(* CoDeSys 2.3.9.59 project: C2_Write_On_USB_or_SD.pro *)
(* Libraries: Standard.lib, Util.lib 20.3.15 10:30:08, SysLibCallback.lib, SysLibSockets.lib, SysLibTasks.lib, SysLibRtc.lib, SysLibFile.lib, SysLibPlcCtrl.lib *)

(* Task configuration *)
TASK tskMain (PRIORITY := 1, INTERVAL := T#20ms);
	MAIN();
END_TASK
TASK tskFiles (PRIORITY := 10, INTERVAL := T#100ms);
	prgCsvLogger();
END_TASK

(* Data type *)
TYPE stParameters :
STRUCT
	Start_stop	: BOOL;
	Temp1		: WORD;
	Temp2		: WORD;
	Temp3		: WORD;
END_STRUCT
END_TYPE

(* POU 10_Program/MAIN, ST *)
PROGRAM MAIN
VAR
	iCpt: INT := 0;
END_VAR
iCpt := iCpt + 1;
END_PROGRAM

(* POU 10_Program/prgCsvLogger, ST *)
PROGRAM prgCsvLogger
VAR
    Horodatage      : DT;					(* Horodate courante *)

    Trig            : R_TRIG;				(* Déclencheur montée *)
    Ligne           : fbStringBuilder;
    Texte           : STRING(255);
    NbOctets        : DWORD;

    xStart			: BOOL;					(* Impulsion externe de création fichier *)
    xDoItDone       : BOOL;					(* Flag interne d'état *)

    FileName        : STRING := '\InternalStorage\log_file.csv'; (* \InternalStorage ou \UsbStorage ou \StorageCard *)
    Fichier         : fbFileWriter;
    Bytes_Written   : DWORD;
    File_Size       : DWORD;
END_VAR
(*=================================================================================================
PROJET          : Data_To_CSV
DESCRIPTION     : Exemple générique de création et d'enregristement de données dans un 
                  fichier .csv stocké dans la mémoire interne du XV100 "/InternalStorage"
---------------------------------------------------------------------------------------------------
MATERIEL CIBLE  : XV102 (Adaptable à d'autres XV/XC en modifiant le path
LOGICIEL        : CODESYS V2.3.9 SP8
LIBRAIRIES      :
	- Standard.lib (V4.10.05) : R_TRIG
	- SysLibFile.lib (V23.9.04) : SysFileOpen, SysFileWrite, SysFileGetSize, SysFileClose

AUTEUR          : COTTANCIN Bruno
DATE            : 24/03/2026
VERSION         : V1.1.0

HISTORIQUE DES MODIFICATIONS :
---------------------------------------------------------------------------------------------------
V1.0.0 | 21/03/2026 | B. COTTANCIN | Création initiale (séquences, function blocks, etc.)
V1.0.1 | 22/03/2026 | B. COTTANCIN | Finalisation de l'architecture générale avant tests
V1.1.0 | 24/03/2026 | B. COTTANCIN | Commentaires FR + en-tête mis à jour

===================================================================================================
IMPORTANT                                 
===================================================================================================
CE PROGRAMME D'ECRITURE CSV DOIT IMPERATIVEMENT ETRE APPELE DANS UNE TACHE SECONDAIRE.

CONFIGURATION RECOMMANDEE : 
- PRIORITE : INFERIEURE A LA TACHE PRINCIPALE (EX: PRIO 10 OU +)           
- TEMPS DE CYCLE : ELEVE (ENVIRON 100MS)                                   

JUSTIFICATION : LES OPERATIONS D'OUVERTURE, D'ECRITURE ET DE FERMETURE DE FICHIER ONT DES ACCES 
MEMOIRE TRES IMPORTANTS. CETTE CONFIGURATION LAISSE LE TEMPS AU SYSTEME DE GERER LES I/O SANS 
PERTURBER LE RYTHME DU PROGRAMME PRINCIPAL (CYCLES RAPIDES).                                      
===================================================================================================

AVERTISSEMENT / DISCLAIMER :
---------------------------------------------------------------------------------------------------
Ce programme est un exemple destiné à valider le fonctionnement de l'application. 
L'utilisateur doit tester ce code dans un environnement sécurisé avant toute mise en production.
Eaton/L'auteur décline toute responsabilité quant à l'exploitation de ce bloc dans une
installation réelle.
=================================================================================================*)


(* Récupération de l'heure système *)
Horodatage := SysRtcGetTime(TRUE);

(* Détection impulsion pour lancer l’écriture *)
Trig(CLK := xStart);

IF Trig.Q AND NOT xDoItDone THEN
    xDoItDone := TRUE;
END_IF;

(* Construction de ligne + écriture fichier CSV *)
IF xDoItDone THEN

    (* Construction de la ligne CSV *)
    Ligne(
        GetTime := Horodatage,
        str_line => Texte,
        length   => NbOctets
    );

    (* Écriture dans le fichier *)
    Fichier(
        adrBuffer        := ADR(Texte),
        strFileName      := FileName,
        dwNumber         := NbOctets,
        xDoItDone        := xDoItDone,
        dwNumber_written => Bytes_Written,
        dwFile_Size      => File_Size
    );
END_IF;
END_PROGRAM

(* POU 20_FunctionBlock/fbStringBuilder, ST *)
FUNCTION_BLOCK fbStringBuilder
VAR_INPUT
	GetTime	: DT;			(* Horodatage du cycle *)
END_VAR

VAR_OUTPUT
    str_line : STRING(255);	(* Ligne CSV générée *)
    length   : INT;			(* Longueur de la ligne *)
END_VAR

VAR
    parameter : stParameters;

    sTime     : STRING(80);
    sT1       : STRING(20);
    sT2       : STRING(20);
    sT3       : STRING(20);

    sCRLF     : STRING := '$0D$0A';
END_VAR
(* Reset de la ligne pour éviter les concat de l'ancien cycle *)
str_line := '';

(* Conversion des données *)
sTime := DT_TO_STRING(GetTime);
sT1   := WORD_TO_STRING(parameter.temp1);
sT2   := WORD_TO_STRING(parameter.temp2);
sT3   := WORD_TO_STRING(parameter.temp3);

(* Nettoyage format date/heure *)
sTime := DELETE(sTime, 4, 0);
sTime := REPLACE(sTime, ' ', 1, 11);

(* Construction de la ligne CSV *)
str_line := CONCAT(str_line, sTime);
str_line := CONCAT(str_line, ';');
str_line := CONCAT(str_line, sT1);
str_line := CONCAT(str_line, ';');
str_line := CONCAT(str_line, sT2);
str_line := CONCAT(str_line, ';');
str_line := CONCAT(str_line, sT3);
str_line := CONCAT(str_line, sCRLF);

(* Longueur de la ligne *)
length := LEN(str_line);
END_FUNCTION_BLOCK

(* POU 20_FunctionBlock/fbFileWriter, ST *)
FUNCTION_BLOCK fbFileWriter
VAR
    FileNumber   : DWORD;
    FileGetSize  : DWORD;
END_VAR

VAR_INPUT
    adrBuffer    : DWORD;
    strFileName  : STRING(80) := 'sauvegarde.csv';
    dwNumber     : DWORD;
END_VAR

VAR_OUTPUT
    dwNumber_written : DWORD;
    dwFile_Size      : DWORD;
END_VAR

VAR_IN_OUT
    xDoItDone : BOOL;
END_VAR
(* Ouverture du fichier en mode ajout *)
FileNumber := SysFileOpen(strFileName, 'a');

IF FileNumber <> 0 THEN
    (* Écriture *)
    SysFileWrite(FileNumber, adrBuffer, dwNumber);

    (* Taille du fichier après écriture *)
    FileGetSize := SysFileGetSize(strFileName);

    (* Fermeture *)
    SysFileClose(FileNumber);

    dwNumber_written := dwNumber;
    dwFile_Size      := FileGetSize;
END_IF

(* Réarmement de l'état *)
xDoItDone := FALSE;
END_FUNCTION_BLOCK

(* POU 10_Program/temp, ST *)
PROGRAM temp
VAR
    Horodatage      : DT;            (* Horodate courante *)

    Trig            : R_TRIG;        (* Détection front montant sur demande visu *)
    fbBuild         : fbStringBuilder;
    sLigne          : STRING(255);
    nNbOctets       : INT;

    xVisu_Start     : BOOL;          (* Commande externe *)
    xWritePending   : BOOL;          (* Flag interne d'autorisation d'écriture *)

    sFileName       : STRING(80) := '\InternalStorage\log_file.csv';
    fbFile          : fbFileWriter;
END_VAR
(* Heure *)
Horodatage := SysRtcGetTime(TRUE);

(* Logique de déclenchement *)
Trig(CLK := xVisu_Start);
IF Trig.Q THEN
 	xWritePending := TRUE;
END_IF;

(* Construction et Écriture (si déclenché) *)
IF xWritePending THEN

	(* Génération de la ligne CSV *)
	fbBuild(GetTime := Horodatage);
	sLigne	:= fbBuild.str_line;
	nNbOctets	:= fbBuild.length;

 	(* Appel du bloc d'écriture *)
	fbFile(
		adrBuffer		:= ADR(sLigne),
 		strFileName	:= sFileName,
		dwNumber	:= INT_TO_DWORD(nNbOctets),
		xDoItDone		:= xWritePending (* Le FB passera xWritePending à FALSE à la fin *)
	);
END_IF;
END_PROGRAM
